// TwinCAT 3 PLC project Untitled1
// ProgramVersion: 3.1.4023.0
// libraries:
//   ESO CCS PLC Simulator Library, * (ccsim)
//   ESO LDC Motor Library, * (ESO)
//   Tc2_Standard, * (Beckhoff Automation GmbH)
//   Tc2_System, * (Beckhoff Automation GmbH)
//   Tc2_Utilities, * (Beckhoff Automation GmbH)
//   Tc3_Module, * (Beckhoff Automation GmbH)
//   VisuDialogs, * (System)
//   ESO LDC Shutter Library,1.1.1.0,ESO
//   VisuSymbols,3.5.10.0,System
// project tree:
//   / GlobalTextList.TcGTLO, PlcTask.TcTTO
//   GVLs/ SCIFY_HMI_Variables.TcGVL
//   POUs/ MAIN.TcPOU
//   VISUs/ SCIFY_Delay_Lines.TcVIS, DL_MOTOR_01_CONFIG.TcVIS, DL_MOTOR_01_CTRL.TcVIS, SCIFY_Cryo.TcVIS, SCIFY_main.TcVIS, VisualizationManager.TcVMO (not stored)
// real-time tasks:
//   TASK PlcTask: cycle T#10ms, priority 20, ADS port 350
// motion (NC):
//   TASK NC-Task 1 SAF: cycle T#2ms, priority 4, ADS port 501
//   TASK NC-Task 1 SVB: cycle T#10ms, priority 8, ADS port 511
//   AXIS DL_Motor_1 (id 2)
//     Dynamic: AccelerationMaximum=2, DecelerationMaximum=2, Acceleration=2, Deceleration=2, Jerk=5
//     Velo: RefSearch=0.5, RefSync=0.5, SlowManual=0.5, FastManual=0.75, Fast=1, Maximum=1.5
//     OtherSettings: AllowMotionCmdToSlave=true, PulseDistancePos=0.5, PulseDistanceNeg=0.5
//     encoder EncType=4
//       EncPara: ScaleFactorNumerator=2.893937e-05, MaxCount=#xffffffff
//         Inc: RefMode=2, RefSoftSyncMask=#x0000ffff
//     drive DrvType=23
//       Analog: VeloReferenz=1.5, TorqueSetpointScale=10, ScaleFactorActTorque=0.1
//       TimeComp: TaskDelayCycles=1
//     controller CtrType=1
//       CtrPara: PriorControlFactor=1
//         PID: PosKp=5
//         Observer: BandWidth=20
//   AXIS Cryo_Motor (id 3)
//     Dynamic: AccelerationMaximum=5, DecelerationMaximum=5, Acceleration=5, Deceleration=5, Jerk=7
//     Velo: RefSearch=0.5, RefSync=0.5, SlowManual=1, FastManual=1, Fast=1.5, Maximum=1.5
//     OtherSettings: AllowMotionCmdToSlave=true, PulseDistancePos=0.5, PulseDistanceNeg=0.5
//     encoder EncType=4
//       EncPara: MaxCount=#xffffffff
//         Inc: RefMode=2, RefSoftSyncMask=#x0000ffff
//     drive DrvType=24
//       Analog: VeloReferenz=1.5, TorqueSetpointScale=10, ScaleFactorActTorque=0.1
//       TimeComp: TaskDelayCycles=1
//     controller CtrType=1
//       CtrPara: PriorControlFactor=1
//         Observer: BandWidth=20
//   AXIS DL_Stepper_Motor_1 (id 4)
//     Dynamic: AccelerationMaximum=1, DecelerationMaximum=1, Acceleration=1, Deceleration=1, Jerk=3
//     Velo: RefSearch=0.1, RefSync=0.1, SlowManual=0.3, FastManual=0.3, Fast=0.1, Maximum=0.4
//     OtherSettings: AllowMotionCmdToSlave=true, PulseDistancePos=0.2, PulseDistanceNeg=0.2
//     encoder EncType=4
//       EncPara: ScaleFactorNumerator=3.051757812e-06, MaxCount=#xffffffff
//         Inc: RefMode=2, RefSoftSyncMask=#x0000ffff
//     drive DrvType=24
//       Analog: VeloReferenz=0.4, TorqueSetpointScale=10, ScaleFactorActTorque=0.1
//       TimeComp: TaskDelayCycles=1
//     controller CtrType=1
//       CtrPara: PriorControlFactor=1
//         Observer: BandWidth=20
// I/O:
//   DEVICE Device 5 (NOV-DP-RAM)
//   DEVICE Device 6 (EtherCAT), AmsNetId 5.83.231.226.7.1
//     Term 10 (EK1100) [EK1100 EtherCAT Coupler (2A E-Bus)]
//       Term 11 (EL7342) [EL7342 2Ch. DC motor output stage (50V, 3.5A)]
//       Term 12 (EL9505) [EL9505 Power supply terminal 5V]
//       Term 13 (EL1124) [EL1124 4Ch. Dig. Input 5V, 10µs, Sensor Power]
//       Term 18 (EL2124) [EL2124 4Ch. Dig. Output 5V, 20mA]
//       Term 11 (EL9011) [EL9011 End Terminal]
//   DEVICE Device 1 (EtherCAT), AmsNetId 5.83.231.226.2.1
//     Term 5 (EK1200) [EK1200-5000 EtherCAT Power supply (2A E-Bus)]
//       Term 6 (EL7047) [EL7047 1Ch. Stepper motor output stage (50V, 5A)]
//       Term 7 (EL2535) [EL2535 2Ch. Pulse Width Current Output (24V, 1A)]
//       Term 8 (EL1084) [EL1084 4Ch. Dig. Input 24V, 3ms, negative]
//       Term 9 (EL2502) [EL2502 2Ch. PWM output, 24V]
//       Term 16 (EL3218) [EL3218-0000 8Ch. Ana. Input PT100 (RTD)]
//       Term 12 (EL9011) [EL9011 End Terminal]
// variable links:
//   NC-Task 1 SAF/Axes/DL_Motor_1 <-> Device 6 (EtherCAT)/Term 10 (EK1100)/Term 11 (EL7342)
//     Drive/Inputs/In/nState1 @bit 3 <-> DCM Status Channel 1/Status/Error
//     Drive/Inputs/In/nState1 @bit 5 <-> DCM Status Channel 1/Status/Moving negative
//     Drive/Inputs/In/nState1 @bit 4 <-> DCM Status Channel 1/Status/Moving positive
//     Drive/Inputs/In/nState1 @bit 1 <-> DCM Status Channel 1/Status/Ready
//     Drive/Inputs/In/nState1 <-> DCM Status Channel 1/Status/Ready to enable
//     Drive/Inputs/In/nState1 @bit 6 <-> DCM Status Channel 1/Status/Torque reduced
//     Drive/Inputs/In/nState1 @bit 2 <-> DCM Status Channel 1/Status/Warning
//     Drive/Inputs/In/nState2 @bit 3 <-> DCM Status Channel 1/Status/Digital input 1
//     Drive/Inputs/In/nState2 @bit 4 <-> DCM Status Channel 1/Status/Digital input 2
//     Drive/Inputs/In/nState2 @bit 5 <-> DCM Status Channel 1/Status/Sync error
//     Drive/Inputs/In/nState2 @bit 7 <-> DCM Status Channel 1/Status/TxPDO Toggle
//     Drive/Inputs/In/nState4 @bit 1 <-> WcState/InputToggle
//     Drive/Inputs/In/nState4 <-> WcState/WcState
//     Drive/Outputs/Out/nCtrl1 <-> DCM Control Channel 1/Control/Enable
//     Drive/Outputs/Out/nCtrl1 @bit 2 <-> DCM Control Channel 1/Control/Reduce torque
//     Drive/Outputs/Out/nCtrl1 @bit 1 <-> DCM Control Channel 1/Control/Reset
//     Drive/Outputs/Out/nCtrl1 @bit 3 <-> DCM Control Channel 1/Control/Threshold active
//     Enc/Inputs/In/nDataIn1 <-> ENC Status Channel 1/Counter value
//     Enc/Inputs/In/nDataIn2 <-> ENC Status Channel 1/Latch value
//     Enc/Inputs/In/nState1 @bit 4 <-> ENC Status Channel 1/Status/Counter overflow
//     Enc/Inputs/In/nState1 @bit 3 <-> ENC Status Channel 1/Status/Counter underflow
//     Enc/Inputs/In/nState1 @bit 7 <-> ENC Status Channel 1/Status/Extrapolation stall
//     Enc/Inputs/In/nState1 @bit 1 <-> ENC Status Channel 1/Status/Latch extern valid
//     Enc/Inputs/In/nState1 @bit 2 <-> ENC Status Channel 1/Status/Set counter done
//     Enc/Inputs/In/nState2 @bit 4 <-> ENC Status Channel 1/Status/Status of extern latch
//     Enc/Inputs/In/nState2 <-> ENC Status Channel 1/Status/Status of input A
//     Enc/Inputs/In/nState2 @bit 1 <-> ENC Status Channel 1/Status/Status of input B
//     Enc/Inputs/In/nState2 @bit 5 <-> ENC Status Channel 1/Status/Sync error
//     Enc/Inputs/In/nState2 @bit 7 <-> ENC Status Channel 1/Status/TxPDO Toggle
//     Enc/Inputs/In/nState4 @bit 1 <-> WcState/InputToggle
//     Enc/Inputs/In/nState4 <-> WcState/WcState
//     Enc/Outputs/Out/nCtrl1 @bit 3 <-> ENC Control Channel 1/Control/Enable latch extern on negative edge
//     Enc/Outputs/Out/nCtrl1 @bit 1 <-> ENC Control Channel 1/Control/Enable latch extern on positive edge
//     Enc/Outputs/Out/nCtrl1 @bit 2 <-> ENC Control Channel 1/Control/Set counter
//     Enc/Outputs/Out/nDataOut1 <-> ENC Control Channel 1/Set counter value
//   Untitled1/Untitled1 Instance <-> Device 1 (EtherCAT)/Term 5 (EK1200)/Term 16 (EL3218)
//     PlcTask Inputs/MAIN.i_TempSensor_{1..4} <-> RTD Inputs Channel {1..4}/Value  (4 links)
//   Untitled1/Untitled1 Instance <-> Device 1 (EtherCAT)/Term 5 (EK1200)/Term 7 (EL2535)
//     PlcTask Inputs/MAIN.Shutter_1.i_nCouplerState <-> InfoData/State
//     PlcTask Outputs/MAIN.iShutterPWM <-> PWM Control Channel 1/PWM output
//   Untitled1/Untitled1 Instance <-> Device 1 (EtherCAT)/Term 5 (EK1200)/Term 8 (EL1084)
//     PlcTask Inputs/MAIN.Shutter_1_Status <-> Channel 1/Input
//   Untitled1/Untitled1 Instance <-> Device 1 (EtherCAT)/Term 5 (EK1200)/Term 9 (EL2502)
//     PlcTask Outputs/MAIN.q_Heater_1 <-> PWM Outputs Channel 1/PWM output
//     PlcTask Outputs/MAIN.q_Heater_2 <-> PWM Outputs Channel 2/PWM output
//   Untitled1/Untitled1 Instance <-> Device 6 (EtherCAT)/Term 10 (EK1100)/Term 11 (EL7342)
//     PlcTask Inputs/MAIN.DL_Motor_01.i_nCouplerState <-> InfoData/State
//   Untitled1/Untitled1 Instance <-> Device 6 (EtherCAT)/Term 10 (EK1100)/Term 13 (EL1124)
//     PlcTask Inputs/MAIN.DL_Motor_01.switches/bLHW <-> Channel 2/Input
//     PlcTask Inputs/MAIN.DL_Motor_01.switches/bUHW <-> Channel 1/Input
//   Untitled1/Untitled1 Instance <-> NC-Task 1 SAF/Axes/DL_Motor_1
//     PlcTask Inputs/MAIN.DL_Motor_01.Axis.NcToPlc <-> Outputs/ToPlc
//     PlcTask Outputs/MAIN.DL_Motor_01.Axis.PlcToNc <-> Inputs/FromPlc

CONFIGURATION Untitled1
    RESOURCE PLC ON TwinCAT3
        TASK PlcTask(INTERVAL := T#10ms, PRIORITY := 20);
        PROGRAM MAIN WITH PlcTask : MAIN;
    END_RESOURCE
END_CONFIGURATION

// ---- GVLs/SCIFY_HMI_Variables.TcGVL
{attribute 'qualified_only'}
VAR_GLOBAL
	

// Temperature Sensors
fTemp_1 : FLOAT;

fTemp_2 : FLOAT;

fTemp_3 : FLOAT;

fTemp_4 : FLOAT;

// Heaters

uiHeater_1 : UINT;
uiHeater_2 : UINT;


END_VAR

// ---- POUs/MAIN.TcPOU
PROGRAM MAIN
VAR

// Motors
DL_Motor_01 : FB_MOTOR;

// Shutters

Shutter_1 : FB_SHUTTER;

Shutter_1_Status AT %I*	 : BOOL;

bIsInitialized			: BOOL	:= FALSE;
	bShutterIsOpen			: BOOL	:= FALSE;
	bShutterButton			: BOOL	:= FALSE;
	iShutterPWM		AT %Q*	: INT	:= 0;
	rShutterVoltage			: REAL;
	sShutterState			: STRING := 'CLOSED';

// Temperature Sensors

i_TempSensor_1 AT %I* : INT;
i_TempSensor_2 AT %I* : INT;
i_TempSensor_3 AT %I* : INT;
i_TempSensor_4 AT %I* : INT;



// Heaters

q_Heater_1 AT %Q* : UINT;
q_Heater_2 AT %Q* : UINT;


END_VAR


DL_Motor_01(sName:='DL_Motor_01', nNOVRAM_DevId:=5, nNOVRAM_Offset:= 1000);

// Shutters

Shutter_1(in_sName:= 'Shutter_1', in_bActiveLowClosed:= TRUE);


IF NOT bIsInitialized THEN

	bIsInitialized := TRUE;
END_IF


IF bShutterButton THEN
	IF NOT bShutterIsOpen THEN
		rShutterVoltage := 24;
	ELSE
		rShutterVoltage := 10;
	END_IF
ELSE
	rShutterVoltage := 0;
END_IF

IF rShutterVoltage > 5 THEN
	bShutterIsOpen := TRUE;
ELSE
	bShutterIsOpen := FALSE;
END_IF

IF bShutterIsOpen THEN
	sShutterState := 'OPEN';
ELSE
	sShutterState := 'CLOSED';
END_IF

iShutterPWM := REAL_TO_INT(32767.0 * rShutterVoltage / 24.0);


// Temperatures
SCIFY_HMI_Variables.fTemp_1 := INT_TO_FLOAT(i_TempSensor_1) /10;
SCIFY_HMI_Variables.fTemp_2 := INT_TO_FLOAT(i_TempSensor_2) /10;
SCIFY_HMI_Variables.fTemp_3 := INT_TO_FLOAT(i_TempSensor_3) /10;
SCIFY_HMI_Variables.fTemp_4 := INT_TO_FLOAT(i_TempSensor_4) /10;

// Heaters
q_Heater_1 := SCIFY_HMI_Variables.uiHeater_1;
q_Heater_2 := SCIFY_HMI_Variables.uiHeater_2;

END_PROGRAM

// ---- GlobalTextList.TcGTLO
TEXTLIST GlobalTextList
  663 = ' °C'
  801 = '%f'
  353 = '%i'
  916 = 'C'
  6 = 'CRYOSTAT'
  165 = 'CRYSTAT'
  379 = 'Delay Lines'
  933 = 'DL_1 Config'
  176 = 'DL_1 Control'
  319 = 'Heater values: 0 OFF and 65535 for Max. PWM'
  978 = 'Heater_1'
  986 = 'Heater_2'
  737 = 'SCIFY Cryostat'
  74 = 'SCIFY Main'
  493 = 'T1'
  848 = 'T2'
  812 = 'T3'
  38 = 'T4'
END_TEXTLIST

// ---- VISUs/SCIFY_Delay_Lines.TcVIS
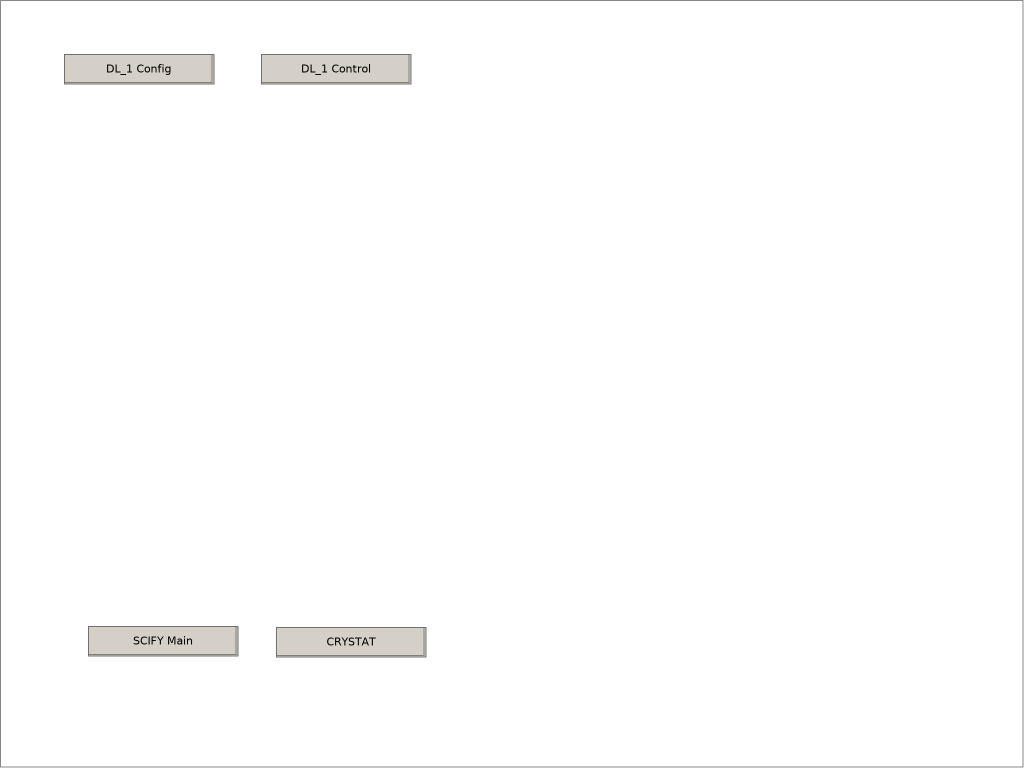
VISUALIZATION SCIFY_Delay_Lines  // 1024x768
    Button (88,626 150x30), "SCIFY Main"
        OnMouseDown: change screen: SCIFY_main
    Button (276,627 150x30), "CRYSTAT"
        OnMouseDown: change screen: SCIFY_Cryo
    Button (64,54 150x30), "DL_1 Config"
        OnMouseDown: change screen: DL_MOTOR_01_CONFIG
    Button (261,54 150x30), "DL_1 Control"
        OnMouseDown: change screen: DL_MOTOR_01_CTRL
END_VISUALIZATION

// ---- VISUs/DL_MOTOR_01_CONFIG.TcVIS
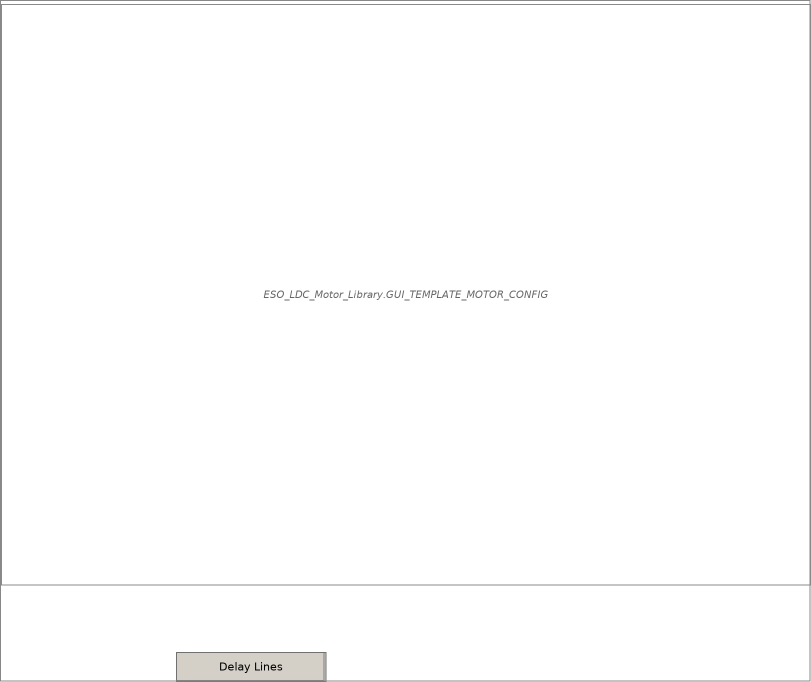
VISUALIZATION DL_MOTOR_01_CONFIG  // 811x682
    Frame (1,4 810x581)
        shows ESO_LDC_Motor_Library.GUI_TEMPLATE_MOTOR_CONFIG(m_Instance := MAIN.DL_Motor_01)
    Button (176,652 150x30), "Delay Lines"
        OnMouseDown: change screen: SCIFY_Delay_Lines
END_VISUALIZATION

// ---- VISUs/DL_MOTOR_01_CTRL.TcVIS
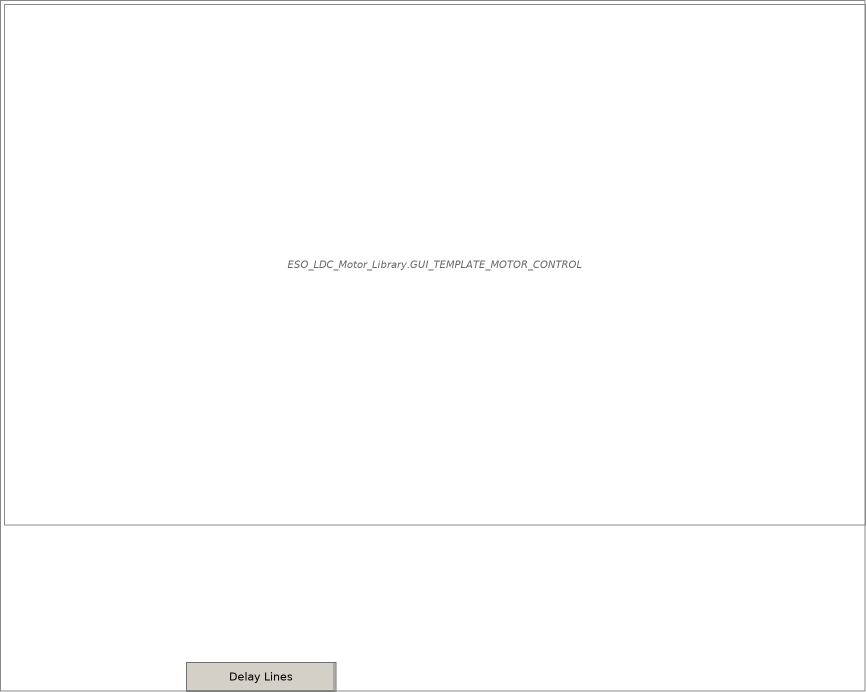
VISUALIZATION DL_MOTOR_01_CTRL  // 866x692
    Frame (4,4 862x521)
        shows ESO_LDC_Motor_Library.GUI_TEMPLATE_MOTOR_CONTROL(m_Instance := MAIN.DL_Motor_01)
    Button (186,662 150x30), "Delay Lines"
        OnMouseDown: change screen: SCIFY_Delay_Lines
END_VISUALIZATION

// ---- VISUs/SCIFY_Cryo.TcVIS
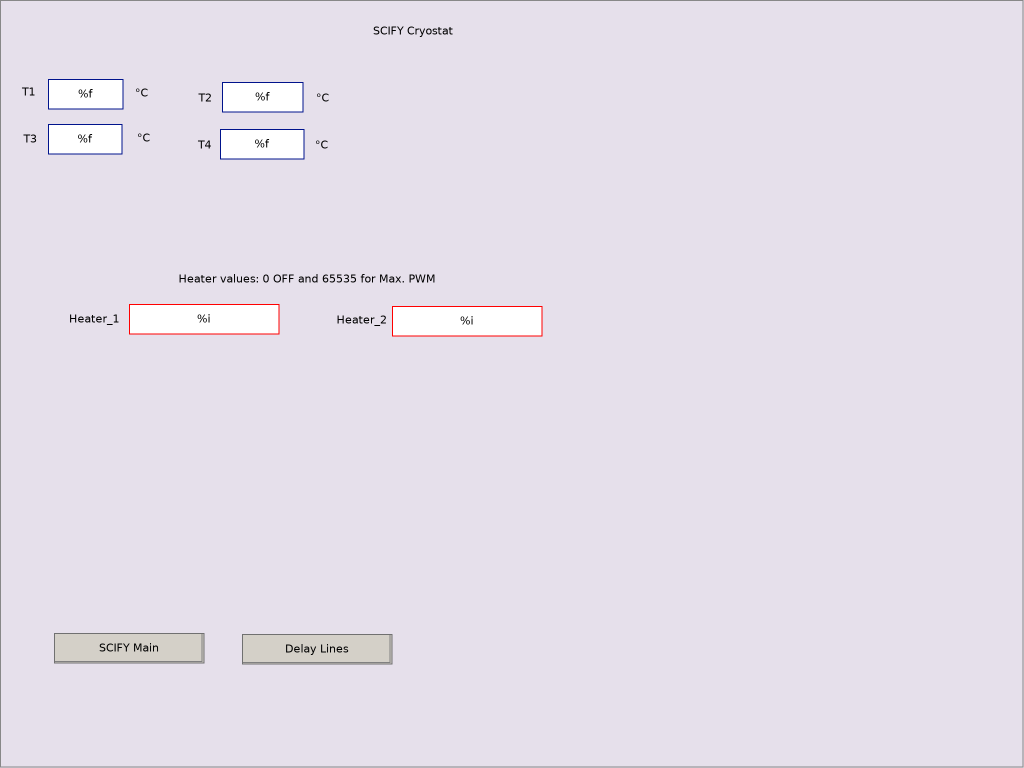
VISUALIZATION SCIFY_Cryo  // 1024x768
    Label (338,6 150x50), "SCIFY Cryostat"
    Textfield (48,79 75x30), "%f", text variable: SCIFY_HMI_Variables.fTemp_1
    Textfield (222,82 81x30), "%f", text variable: SCIFY_HMI_Variables.fTemp_2
    Textfield (48,124 74x30), "%f", text variable: SCIFY_HMI_Variables.fTemp_3
    Textfield (220,129 84x30), "%f", text variable: SCIFY_HMI_Variables.fTemp_4
    Textfield (129,304 150x30), "%i", text variable: SCIFY_HMI_Variables.uiHeater_1
        OnMouseClick: write the text variable via VisuDialogs.Numpad, min 0, max 65535
    Textfield (392,306 150x30), "%i", text variable: SCIFY_HMI_Variables.uiHeater_2
        OnMouseClick: write the text variable via VisuDialogs.Numpad, min 0, max 65535
    Label (19,77 20x30), "T1"
    Label (191,83 29x30), "T2"
    Label (19,124 23x30), "T3"
    Label (196,130 18x30), "T4"
    Label (64,304 61x30), "Heater_1"
    Label (335,305 54x30), "Heater_2"
    Label (122,78 36x30), "°C"
    Label (303,83 36x30), "°C"
    Label (124,123 36x30), "°C"
    Label (302,130 36x30), "°C"
    Label (65,264 484x30), "Heater values: 0 OFF and 65535 for Max. PWM"
    Button (54,633 150x30), "SCIFY Main"
        OnMouseDown: change screen: SCIFY_main
    Button (242,634 150x30), "Delay Lines"
        OnMouseDown: change screen: SCIFY_Delay_Lines
END_VISUALIZATION

// ---- VISUs/SCIFY_main.TcVIS
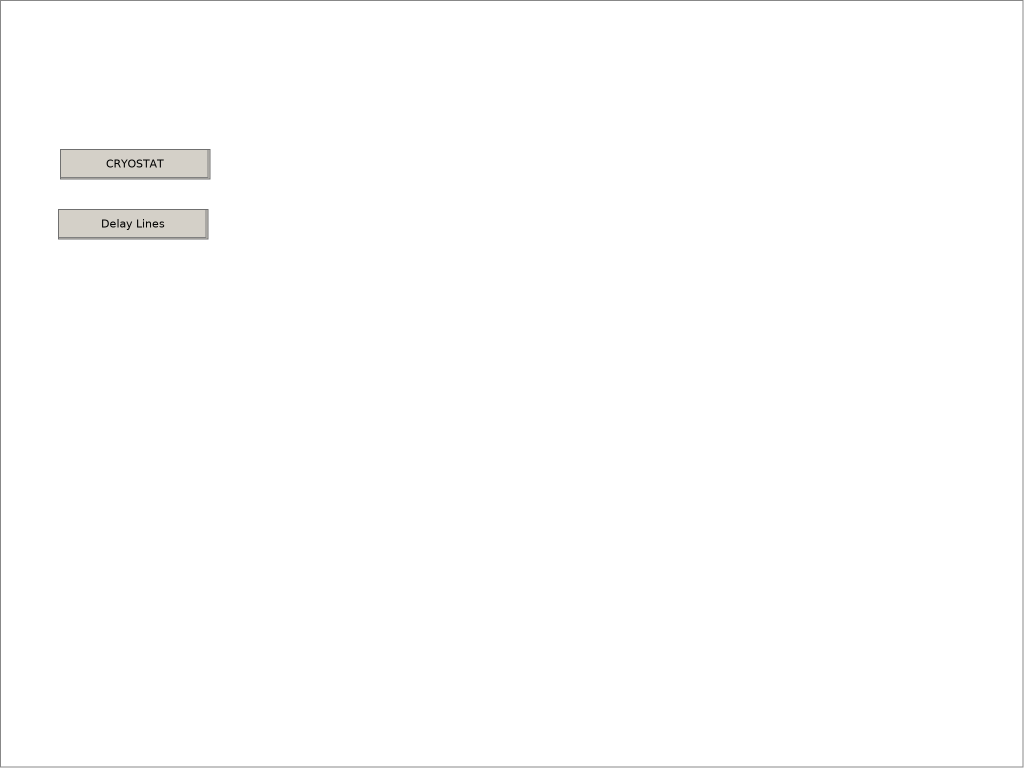
VISUALIZATION SCIFY_main  // 1024x768
    Button (60,149 150x30), "CRYOSTAT"
        OnMouseDown: change screen: SCIFY_Cryo
    Button (58,209 150x30), "Delay Lines"
        OnMouseDown: change screen: SCIFY_Delay_Lines
END_VISUALIZATION
